TYPE ST_NciChannel_Ref :
STRUCT
  NcToPlc AT %I*: NcToPlc_NciChannel_Ref;   //  Externer Datentyp!
  PlcToNc AT %Q*: PlcToNc_NciChannel_Ref;   //  Externer Datentyp!
END_STRUCT
END_TYPE

(* stored: Version 1.1.0.1, ProductVersion 3.1.4024.9
   DUT ST_NciChannel_Ref: Id {45452d2b-5996-0ee1-1adc-7cf3d4675fa6} *)
